FUNCTION_BLOCK AXE_plant (* Basic Function Block Type *)
  (* Standard: 61499-2 *)
  (* Version 0.0, 13/06/2022, Etienne, Schneider Electric, Template *)
  PACKAGE Main;
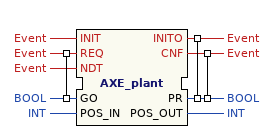
  EVENT_INPUT
    INIT; (* Initialization Request *)
    REQ WITH GO; (* Normal Execution Request *)
    NDT;
  END_EVENT
  EVENT_OUTPUT
    INITO WITH PR; (* Initialization Confirm *)
    CNF WITH PR; (* Execution Confirmation *)
  END_EVENT
  VAR_INPUT
    GO : BOOL;
    POS_IN : INT;
  END_VAR
  VAR_OUTPUT
    PR : BOOL;
    POS_OUT : INT;
  END_VAR
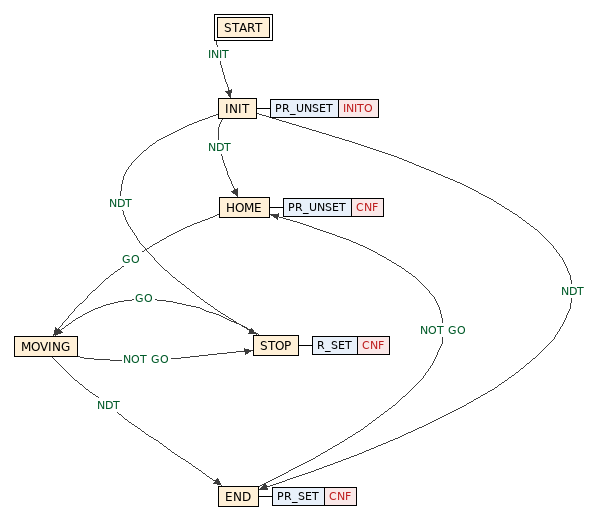
  EC_STATES
    START; (* Initial State *)
    HOME : PR_UNSET -> CNF;
    MOVING;
    END : PR_SET -> CNF;
    INIT : PR_UNSET -> INITO;
    STOP : R_SET -> CNF;
  END_STATES
  EC_TRANSITIONS
    HOME TO MOVING := GO;
    MOVING TO END := NDT;
    INIT TO HOME := NDT;
    INIT TO END := NDT;
    START TO INIT := INIT;
    END TO HOME := NOT GO;
    MOVING TO STOP := NOT GO;
    STOP TO MOVING := GO;
    INIT TO STOP := NDT;
  END_TRANSITIONS
  ALGORITHM PR_SET IN ST:
;
PR:=TRUE;
POS_OUT:=POS_IN;
  END_ALGORITHM
  ALGORITHM PR_UNSET IN ST:
;
PR := FALSE;
  END_ALGORITHM
  ALGORITHM R_SET IN ST:
POS_OUT:=5;
  END_ALGORITHM
END_FUNCTION_BLOCK
